(* PLC project recipe, Dassault Systèmes ControlBuild 2024x Refresh1 *)
(* stored: creationDateTime 2024-04-12T14:05:56-01:00 *)

FUNCTION_BLOCK copie_batch.recipe
  VAR_OUTPUT
    flourWeight : DINT := 0;
  END_VAR
  VAR_OUTPUT
    syrup1Weight : DINT := 0;
    syrup2Weight : DINT := 0;
    syrup3Weight : DINT := 0;
  END_VAR
  VAR CONSTANT
    recipeNumber : DINT := 1;
  END_VAR

CASE recipeNumber OF
	1 :
		flourWeight := 200;
		syrup1Weight := 150;
		syrup2Weight := 100;
		syrup3Weight := 50;
	2 :
		flourWeight := 200;
		syrup1Weight := 50;
		syrup2Weight := 150;
		syrup3Weight := 100;
	3 :
		flourWeight := 200;
		syrup1Weight := 50;
		syrup2Weight := 100;
		syrup3Weight := 150;
	
END_CASE;
END_FUNCTION_BLOCK
